{attribute 'qualified_only'}
{attribute 'strict'}
TYPE E_SimulatorStates :
(
	Run,
	Stop
);
END_TYPE

(* stored: Version 1.1.0.1, ProductVersion 3.1.4024.12
   DUT E_SimulatorStates: Id {c69b4365-993b-4254-b587-4c20748b81d7} *)
